INTERFACE I_EventHandler

METHOD PUBLIC HandleEvent
VAR_INPUT
	Event : I_Event;
END_VAR
END_METHOD

END_INTERFACE

(* stored: Version 1.1.0.1, ProductVersion 3.1.4024.12
   Itf I_EventHandler: Id {53aefc50-912d-481b-b2d1-1c8b280e315b}
   Method HandleEvent: Id {31f1d8e0-0021-4c9e-beaf-9765834bc18f} *)
